{attribute 'qualified_only'}
{attribute 'strict'}
{attribute 'to_string'}
TYPE E_DriveControl : (
		Idle := 0,
		Activate_auto_mode,
		Activate_supervisor_error,
		Activate_manual_mode,
		Activate_emergency_stop
	) UINT;
END_TYPE

(* stored: Version 1.1.0.1
   DUT E_DriveControl: Id {2c489590-5ba0-4f71-996f-2df7f8433b0a} *)
